// TIA Portal V16 export
// export: Created 2026-04-03T07:10:44.6628572Z, ExportSetting WithDefaults, DisplayName Totally Integrated Automation Portal, DisplayVersion V16, DisplayName TIA Portal Version Control Interface, DisplayVersion V16, DisplayName TIA Portal Openness, DisplayVersion V16, DisplayName STEP 7 Professional, DisplayVersion V16, DisplayName STEP 7 Safety, DisplayVersion V16, DisplayName WinCC Advanced, DisplayVersion V16
VAR_GLOBAL   // PLC tag table "Tag tanks"
END_VAR
VAR_GLOBAL CONSTANT   // user constants
   c_Count_TRN : Int := 3;
   c_Count_POL : Int := 10;
   c_Count_BUL : Int := 4;
   c_Count_MOL : Int := 12;
END_VAR
